PROGRAM PRG_1_PlcTask
VAR
//fbLogHandler: FB_LogHandler;
	// PRG_DCCM_MONO: INT;
END_VAR

PRG_DCCM_MONO();
//fbLogHandler();

END_PROGRAM

(* stored: Version 1.1.0.1, ProductVersion 3.1.4024.12
   POU PRG_1_PlcTask: Id {21f3a158-4837-47ff-8ec7-29454a44967d}, SpecialFunc None *)
